FUNCTION_BLOCK FB_Linked_List_Queue IMPLEMENTS I_Queue
VAR
	fbLinked_List : FB_Singly_Linked_List;
END_VAR

(* Removes element from the front of the queue. *)
METHOD Dequeue : T_DATA_TYPE
Dequeue := THIS^.fbLinked_List.Pop();
END_METHOD

(* Empties/Clears/Deletes all elements on the stack. *)
METHOD Empty
THIS^.fbLinked_List.Empty();
END_METHOD

(* Adds element to the rear of the queue. *)
METHOD Enqueue
VAR_INPUT
	Data	: T_DATA_TYPE;
END_VAR
THIS^.fbLinked_List.Create(Data);
END_METHOD

METHOD FB_exit : BOOL
VAR_INPUT
	(* if TRUE, the exit method is called for exiting an instance that is copied afterwards (online change).*)
	bInCopyCode	: BOOL;
END_VAR
THIS^.Empty();
END_METHOD

METHOD FB_init : BOOL
VAR_INPUT
	(* if TRUE, the retain variables are initialized (warm start / cold start)*)
	bInitRetains	: BOOL;
	(* if TRUE, the instance afterwards gets moved into the copy code (online change)*)
	bInCopyCode	: BOOL;
END_VAR
END_METHOD

(* Checks of queue is empty. *)
METHOD Is_Empty : BOOL
Is_Empty := THIS^.fbLinked_List.Is_Empty();
END_METHOD

(* Gets element at any position of the queue, without removing it.*)
METHOD Peek : T_DATA_TYPE
VAR_INPUT
	nPosition	: DINT;
END_VAR
Peek := THIS^.fbLinked_List.Peek(nPosition);
END_METHOD

(* Traverse the queue and display each element as an array. *)
METHOD Show
VAR_IN_OUT
	aList :  ARRAY[*] OF T_DATA_TYPE; // Array to display data in list.
END_VAR
THIS^.fbLinked_List.Show(aList);
END_METHOD

(* Gets size of the queue. *)
METHOD Size : DINT
Size := THIS^.fbLinked_List.Size();
END_METHOD

END_FUNCTION_BLOCK

(* stored: Version 1.1.0.1, ProductVersion 3.1.4024.4
   POU FB_Linked_List_Queue: Id {4f1203bd-4461-4bf6-ac1b-1010eb6cd6fc}, SpecialFunc None
   Method Dequeue: Id {36c56a29-2008-43aa-98cc-8681eb03c4e3}
   Method Empty: Id {89bb4ed3-660e-49e6-acbd-cebec57cbf22}
   Method Enqueue: Id {8bbe41d5-5089-43fe-940b-a83ea299e3c0}
   Method FB_exit: Id {562b1a94-f54e-420c-9e12-225a42181e14}
   Method FB_init: Id {93113c57-65f1-4df7-8747-8bbe258cdc94}
   Method Is_Empty: Id {ccc19132-53e2-4f82-b091-7fd31c79ed4e}
   Method Peek: Id {002c8ba8-ddf7-458f-a558-b892ba1f6a39}
   Method Show: Id {a894857c-ef29-4206-bcd0-db8721199075}
   Method Size: Id {24bb2dc8-1984-401c-927f-bd9b3255464e} *)
